ADAPTER AStorage (* Adapter Interface *)
  (* Standard: 61499-1 *)
  (* Version 1.0, 2021-09-15, dorofeev *)
  (* Compiler header: package fb.test; *)
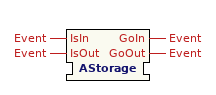
  EVENT_INPUT
    IsIn; (* Request from Socket *)
    IsOut; (* Response from Socket *)
  END_EVENT
  EVENT_OUTPUT
    GoIn; (* Confirmation from Plug *)
    GoOut;
  END_EVENT
  SERVICE PLUG/SOCKET (* Adapter Interface *)
    SEQUENCE request_confirm
      SOCKET.REQ(REQD) -> PLUG.REQ(REQD);
      PLUG.CNF(CNFD) -> SOCKET.CNF(CNFD);
    END_SEQUENCE
    SEQUENCE indication_response
      PLUG.IND(INDD) -> SOCKET.IND(INDD);
      SOCKET.RSP(RSPD) -> PLUG.RSP(RSPD);
    END_SEQUENCE
  END_SERVICE
END_ADAPTER
